TYPE HMI_MAN_TemplateClean :
STRUCT

END_STRUCT
END_TYPE

(* stored: Version 1.1.0.1
   DUT HMI_MAN_TemplateClean: Id {9d60cffa-578b-4745-afa9-049f24ef55a2} *)
